GLOBALCONSTANTS IG5_NAME_Functions (* Industry Group 5 specific function defines *)
  (* Standard: 61499-1 *)
  (* Version 1.0, 2026-06-29, Franz Höpfinger, Demmler Andreas Fahrzeugbau *)
  PACKAGE isobus::pgn::const;
  VAR_GLOBAL CONSTANT
    F_INDUSTRIAL_GEN_SET_SUPPLEMENTAL_ENGINE_CONTROL_SENSING : BYTE := 128; (* Sys: Industrial-Process Control-Stationary (Gen-Sets), Func: Supplemental Engine Control Sensing *)
    F_INDUSTRIAL_GEN_SET_GENERATOR_SET_CONTROLLER : BYTE := 129; (* Sys: Industrial-Process Control-Stationary (Gen-Sets), Func: Generator Set Controller - Generator *)
    F_INDUSTRIAL_GEN_SET_GENERATOR_VOLTAGE_REGULATOR : BYTE := 130; (* Sys: Industrial-Process Control-Stationary (Gen-Sets), Func: Generator Voltage Regulator *)
    F_INDUSTRIAL_GEN_SET_CHOKE_ACTUATOR : BYTE := 131; (* Sys: Industrial-Process Control-Stationary (Gen-Sets), Func: Choke Actuator - Device used to *)
    F_WELL_STIMULATION_PUMP : BYTE := 132; (* Sys: , Func: Well Stimulation Pump - Device which communicates operating parameters of a well *)
    F_INDUSTRIAL_GEN_SET_NOT_AVAILABLE : BYTE := 255; (* Sys: Industrial-Process Control-Stationary (Gen-Sets), Func: Not Available - This assignment can *)
    F_NOT_AVAILABLE : BYTE := 255; (* Sys: Not Available, Func: Not Available - This assignment can be used until an explicit function *)
  END_VAR
END_GLOBALCONSTANTS
